FUNCTION "addMessageInfo" : Void
{ S7_Optimized_Access := 'TRUE' }
VERSION : 0.1
   VAR_INPUT
      msg : WString;
   END_VAR


BEGIN
	(*
	--> UnitTest: Add new info message
	*)

	IF "DB_UnitTest".index < "arraySize"("DB_UnitTestControl".msg) THEN
	    "DB_UnitTestControl".msg["DB_UnitTest".index] := #msg;
	    "DB_UnitTest".index += UINT#1;
	ELSE
	    "DB_UnitTestControl".msg["arraySize"("DB_UnitTestControl".msg)] := WSTRING#'limit of messages array reached';
	END_IF;


END_FUNCTION

